FUNCTION_BLOCK FB_TrafficLight IMPLEMENTS ITrafficLight
VAR
	_state : E_LightState := E_LightState.Red;
END_VAR

{warning 'add property implementation'}
PROPERTY CurrentState : E_LightState
GET
CurrentState := _state;
END_GET
END_PROPERTY

METHOD PUBLIC RequestGreen
VAR_INPUT
END_VAR
_state := E_LightState.Green;
END_METHOD

END_FUNCTION_BLOCK

(* stored: Version 1.1.0.1, ProductVersion 3.1.4024.12
   POU FB_TrafficLight: Id {8be2b364-8d2f-4ca1-a6a3-b8591690800c}, SpecialFunc None
   Property CurrentState: Id {946b4ff7-ea0d-42b1-93f6-cca405deadaf}
   Get Get: Id {d7cf4dc2-ada4-4975-91df-ca5b74d507fe}
   Method RequestGreen: Id {7eadf869-ec5e-4e0c-9426-0678f3962762} *)
